(*

short summary
=================
This interface provides assert statements for Windows-1252 and Windows-1251 string pointers

.. attention:: 
	All strings are handled as null-terminated byte streams

.. <legal notes>

legal notes
=================
| SPDX-FileCopyrightText: © 2024 ekvip automation GmbH <info@ekvip.de>
| SPDX-License-Identifier: Apache-2.0
| For details check: Apache-2.0_

.. _Apache-2.0: https://www.apache.org/licenses/LICENSE-2.0

.. </legal notes>

methods
==================

*)

INTERFACE INTERNAL IWindows125xStringPointerAssertions EXTENDS IAssertCallBackSetter

(*

short summary
=================
This assertion method checks if the current string ``stringToCheck`` contains the search string ``searchString``

.. attention:: 
	All strings are handled as null-terminated byte streams

.. <legal notes>

legal notes
=================
| SPDX-FileCopyrightText: © 2024 ekvip automation GmbH <info@ekvip.de>
| SPDX-License-Identifier: Apache-2.0
| For details check: Apache-2.0_

.. _Apache-2.0: https://www.apache.org/licenses/LICENSE-2.0

.. </legal notes>

parameters
=================

*)

METHOD contains : IWindows125xStringPointerAssertions
VAR_INPUT
	(* current string to check *)
	stringToCheck	:POINTER TO BYTE;
	(* string must be found in ``stringToCheck`` *)
	searchString	:POINTER TO BYTE;
	(* ``TRUE`` means ignore cases; ``FALSE`` means that cases must be equal too *)
	ignoreCases		:BOOL;
	(* message if the assertion is false *)
	message			:AssertMessage;
END_VAR
END_METHOD

(*

short summary
=================
This assertion method checks if the current string ``stringToCheck`` doesn't contain the search string ``searchString``

.. attention:: 
	All strings are handled as null-terminated byte streams

.. <legal notes>

legal notes
=================
| SPDX-FileCopyrightText: © 2022 ekvip automation GmbH <info@ekvip.de>
| SPDX-License-Identifier: Apache-2.0
| For details check: Apache-2.0_

.. _Apache-2.0: https://www.apache.org/licenses/LICENSE-2.0

.. </legal notes>

parameters
=================

*)

METHOD containsNo : IWindows125xStringPointerAssertions
VAR_INPUT
	(* current string to check *)
	stringToCheck	:POINTER TO BYTE;
	(* string must be found in ``stringToCheck`` *)
	searchString	:POINTER TO BYTE;
	(* ``TRUE`` means ignore cases; ``FALSE`` means that cases must be equal too *)
	ignoreCases		:BOOL;
	(* message if the assertion is false *)
	message			:AssertMessage;
END_VAR
END_METHOD

(*

short summary
=================
This assertion method checks if the current string ``stringToCheck`` ends with the string ``end``

.. attention:: 
	All strings are handled as null-terminated byte streams

.. <legal notes>

legal notes
=================
| SPDX-FileCopyrightText: © 2022 ekvip automation GmbH <info@ekvip.de>
| SPDX-License-Identifier: Apache-2.0
| For details check: Apache-2.0_

.. _Apache-2.0: https://www.apache.org/licenses/LICENSE-2.0

.. </legal notes>

parameters
=================

*)

METHOD endsWith : IWindows125xStringPointerAssertions
VAR_INPUT
	(* current string to check *)
	stringToCheck	:POINTER TO BYTE;
	(* string must be the end of ``stringToCheck`` *)
	end				:POINTER TO BYTE;
	(* ``TRUE`` means ignore cases; ``FALSE`` means that cases must be equal too *)
	ignoreCases		:BOOL;
	(* ``TRUE`` means truncation of spaces on the right side of ``stringToCheck``*)
	trimRight		:BOOL;
	(* message if the assertion is false *)
	message			:AssertMessage;
END_VAR
END_METHOD

(*

short summary
=================
This assertion method checks if the current string ``stringToCheck`` is equal to ``expected``

.. attention:: 
	All strings are handled as null-terminated byte streams

.. <legal notes>

legal notes
=================
| SPDX-FileCopyrightText: © 2022 ekvip automation GmbH <info@ekvip.de>
| SPDX-License-Identifier: Apache-2.0
| For details check: Apache-2.0_

.. _Apache-2.0: https://www.apache.org/licenses/LICENSE-2.0

.. </legal notes>

parameters
=================

*)

METHOD isEqualTo : IWindows125xStringPointerAssertions
VAR_INPUT
	(* current string to check *)
	stringToCheck	:POINTER TO BYTE;
	(* ``stringToCheck`` must be equal to expected *)
	expected		:POINTER TO BYTE;
	(* ``TRUE`` means ignore cases; ``FALSE`` means that cases must be equal too *)
	ignoreCases		:BOOL;
	(* message if the assertion is false *)
	message			:AssertMessage;
END_VAR
END_METHOD

(*

short summary
=================
This assertion method checks if the current string ``stringToCheck`` is not equal to ``unexpected``

.. attention:: 
	All strings are handled as null-terminated byte streams

.. <legal notes>

legal notes
=================
| SPDX-FileCopyrightText: © 2022 ekvip automation GmbH <info@ekvip.de>
| SPDX-License-Identifier: Apache-2.0
| For details check: Apache-2.0_

.. _Apache-2.0: https://www.apache.org/licenses/LICENSE-2.0

.. </legal notes>

parameters
=================

*)

METHOD isNotEqualTo : IWindows125xStringPointerAssertions
VAR_INPUT
	(* current string to check *)
	stringToCheck	:POINTER TO BYTE;
	(* ``stringToCheck`` must be not equal to expected *)
	unexpected		:POINTER TO BYTE;
	(* ``TRUE`` means ignore cases; ``FALSE`` means that cases must be equal too *)
	ignoreCases		:BOOL;
	(* message if the assertion is false *)
	message			:AssertMessage;
END_VAR
END_METHOD

(*

short summary
=================
This assertion method checks if the current string ``stringToCheck`` length is equal to ``expectedLength``

.. attention:: 
	All strings are handled as null-terminated byte streams

.. <legal notes>

legal notes
=================
| SPDX-FileCopyrightText: © 2022 ekvip automation GmbH <info@ekvip.de>
| SPDX-License-Identifier: Apache-2.0
| For details check: Apache-2.0_

.. _Apache-2.0: https://www.apache.org/licenses/LICENSE-2.0

.. </legal notes>

parameters
=================

*)

METHOD lenghtIsExact : IWindows125xStringPointerAssertions
VAR_INPUT
	(* current string to check *)
	stringToCheck	:POINTER TO BYTE;
	(* expected length of ``stringToCheck`` *)
	expectedLength	:UDINT;
	(* message if the assertion is false *)
	message			:AssertMessage;
END_VAR
END_METHOD

(*

short summary
=================
This assertion method checks if the current string ``stringToCheck`` length is equal or less than to ``maxLength``

.. attention:: 
	All strings are handled as null-terminated byte streams

.. <legal notes>

legal notes
=================
| SPDX-FileCopyrightText: © 2022 ekvip automation GmbH <info@ekvip.de>
| SPDX-License-Identifier: Apache-2.0
| For details check: Apache-2.0_

.. _Apache-2.0: https://www.apache.org/licenses/LICENSE-2.0

.. </legal notes>

parameters
=================

*)

METHOD lenghtIsMax : IWindows125xStringPointerAssertions
VAR_INPUT
	(* current string to check *)
	stringToCheck	:POINTER TO BYTE;
	(* upper limit of the length of ``stringToCheck`` *)
	maxLength		:UDINT;
	(* message if the assertion is false *)
	message			:AssertMessage;
END_VAR
END_METHOD

(*

short summary
=================
This assertion method checks if the current string ``stringToCheck`` length is equal or grater than to ``minLength``

.. attention:: 
	All strings are handled as null-terminated byte streams

.. <legal notes>

legal notes
=================
| SPDX-FileCopyrightText: © 2022 ekvip automation GmbH <info@ekvip.de>
| SPDX-License-Identifier: Apache-2.0
| For details check: Apache-2.0_

.. _Apache-2.0: https://www.apache.org/licenses/LICENSE-2.0

.. </legal notes>

parameters
=================

*)

METHOD lenghtIsMin : IWindows125xStringPointerAssertions
VAR_INPUT
	(* current string to check *)
	stringToCheck	:POINTER TO BYTE;
	(* lower limit of the length of ``stringToCheck`` *)
	minLength		:UDINT;
	(* message if the assertion is false *)
	message			:AssertMessage;
END_VAR
END_METHOD

(*

short summary
=================
This assertion method checks if the current string ``stringToCheck`` length is between ``minLenght`` and ``maxLenght``

.. attention:: 
	All strings are handled as null-terminated byte streams

.. <legal notes>

legal notes
=================
| SPDX-FileCopyrightText: © 2022 ekvip automation GmbH <info@ekvip.de>
| SPDX-License-Identifier: Apache-2.0
| For details check: Apache-2.0_

.. _Apache-2.0: https://www.apache.org/licenses/LICENSE-2.0

.. </legal notes>

parameters
=================

*)

METHOD lengthIsBetween : IWindows125xStringPointerAssertions
VAR_INPUT
	(* current string to check *)
	stringToCheck	:POINTER TO BYTE;
	(* lower limit of the string length *)
	minLenght		:UDINT;
	(* upper limit of the string length *)
	maxLenght		:UDINT;
	(* message if the assertion is false *)
	message			:AssertMessage;
END_VAR
END_METHOD

(*

short summary
=================
This assertion method checks if the current string ``stringToCheck`` starts with string ``start``

.. attention:: 
	All strings are handled as null-terminated byte streams

.. <legal notes>

legal notes
=================
| SPDX-FileCopyrightText: © 2022 ekvip automation GmbH <info@ekvip.de>
| SPDX-License-Identifier: Apache-2.0
| For details check: Apache-2.0_

.. _Apache-2.0: https://www.apache.org/licenses/LICENSE-2.0

.. </legal notes>

parameters
=================

*)

METHOD startsWith : IWindows125xStringPointerAssertions
VAR_INPUT
	(* current string to check *)
	stringToCheck	:POINTER TO BYTE;
	(* expected start of ``stringToCheck`` *)
	start			:POINTER TO BYTE;
	(* ``TRUE`` means ignore cases; ``FALSE`` means that cases must be equal too *)
	ignoreCases		:BOOL;
	(* ``TRUE`` means truncation of spaces on the left side of ``stringToCheck``*)
	trimLeft		:BOOL;
	(* message if the assertion is false *)
	message			:AssertMessage;
END_VAR
END_METHOD

END_INTERFACE

(* stored: Version 1.1.0.1, ProductVersion 3.1.4024.12
   Itf IWindows125xStringPointerAssertions: Id {e1bedbfd-01d3-4166-b1b8-0848edc60fdd}
   Method contains: Id {ca20ac10-f042-4124-8916-4171e9d663e5}
   Method containsNo: Id {8c632835-cbdf-4c3a-aa02-463682a3b496}
   Method endsWith: Id {b8f179c5-571d-4e1f-b2db-bcc807b1c75b}
   Method isEqualTo: Id {b6d6750a-211f-427f-a287-2cf7aa6463ef}
   Method isNotEqualTo: Id {300067c5-ab62-49c9-957e-876265bae97b}
   Method lenghtIsExact: Id {256b6148-f5fd-4b0e-9462-11e94f7c200e}
   Method lenghtIsMax: Id {42050223-4c15-4f15-8330-8b472c546878}
   Method lenghtIsMin: Id {a18751a4-7a1d-4349-8321-9461830c290b}
   Method lengthIsBetween: Id {dc284354-2443-4d8e-86d6-0fbf84e047fe}
   Method startsWith: Id {6bd1fa7c-5fb8-4340-86bb-ccf6b801b201} *)
